# EPICS autosave request: autosave/galil_profileMoveAxis.req
$(P)$(R):M$(M)MoveMode
